FUNCTION_BLOCK InputOutputConvert
VAR_INPUT
END_VAR
VAR_OUTPUT
END_VAR
VAR
END_VAR


//Inputs
LevelMeter := (WORD_TO_INT(InputWordArea[0])*300)/1000;
FlowMeter  := (WORD_TO_INT(InputWordArea[1])*300)/1000;
SetPoint   := (WORD_TO_INT(InputWordArea[2])*300)/1000;
//Outputs
OutputWordArea[0] := INT_TO_WORD(FillValve);
OutputWordArea[1] := INT_TO_WORD(DischargeValve);
SP		   := SetPoint;
OutputWordArea[2] := INT_TO_WORD(SP);
PV		   := LevelMeter;
OutputWordArea[3] := INT_TO_WORD(PV);

//
Start := InputBitArea[0].0;
Reset := InputBitArea[0].1;
Stop  := InputBitArea[0].2;
//
OutputBitArea[0].0 := StartLight;
OutputBitArea[0].1 := ResetLight;
OutputBitArea[0].2 := StopLight;

END_FUNCTION_BLOCK

(* stored: Version 1.1.0.1, ProductVersion 3.1.4024.6
   POU InputOutputConvert: Id {1c806a45-2259-462f-848e-cfc9e3acb681}, SpecialFunc None *)
